(* Logix 5000 project; controller BTS01 vendor 1 type 14 code 217 rev 32.14; software revision 32.04; part 11 of 15 *)
(* tags used below, declared in another part *)
   AG1101 : DTE_VFD;   // Tank 1100 Agitator
   AG1101_CIP_ENABLE : BOOL;
   AG1201 : DTE_VFD;   // Tank 1200 Agitator
   AG1201_CIP_ENABLE : BOOL;
   C02S01 : REAL[8];   // 5069-IF8
   C02S03 : INT;   // 5069-IB16
   C02S06 : INT;   // 5069-IB16
   CAUSTIC1_TIME_REM : DINT;   // CIP 1 CAUSTIC TIM REMAINING
   CIP1_SUPPLY_TEMP_OFFSET : DINT;   // CIP 1 SUPPLY TEMP OFFSET FROM RETURN TEMP SETPOINT
   CIP_1_ACTIVE_CIRCUIT : DINT;
   CIP_1_ACTIVE_PROGRAM : CIP_PROGRAM;
   CIP_1_ACTIVE_STEP : CIP_STEP_DEF;   // CIP 1 ACTIVE STEP DATA
   CIP_1_ACTIVE_STEP_NUMBER : DINT;
   CIP_1_ACTIVE_STEP_SUP_TEMP : DINT;   // CIP 1 SUPPLY TEMP SETPOINT FOR ACTIVE STEP
   CIP_1_ACTIVE_STEP_TIME : DINT;
   CIP_1_ALARM_INDICATOR : DINT;   // ALARM STATE INDICATOR AT HMI
   CIP_1_ALARMS : DINT[30];
   CIP_1_CAUSTIC_TRANS_ACT : BOOL;   // CIP 1 RETURN TO CAUSTIC TANK LEVEL TRANSITION ACTIVE
   CIP_1_CIRCUIT_SELECT_HMI : INT;
   CIP_1_CURRENT_STEP_MESSAGE_INT : DINT;
   CIP_1_FLOW_PROOF : BOOL;   // CIP 1 FLOW PROOF BIT 0 = NO FLOW 1 = FLOW
   CIP_1_HOLD_LATCH : BOOL;
   CIP_1_HOLD_PB_CTU : COUNTER;
   CIP_1_HOLD_PB_HMI : BOOL;
   CIP_1_HOLD_TIME : REAL;
   CIP_1_LOAD_ACTIVE_CIP_RECIPE_PB : BOOL;
   CIP_1_OPERATOR_ACK : BOOL;   // CIP 1 SEQUENCER OPERATOR ACKNOWLEDGE
   CIP_1_OPERATOR_ACK_PB_HMI : BOOL;
   CIP_1_PRERINSE_TRANS_ACT : BOOL;   // CIP 1 RETURN TO PRERINSE TANK LEVEL TRANSITION ACTIVE
   CIP_1_PROGRAMS : CIP_PROGRAM[30];
   CIP_1_RECIPE_SELECTED_HMI : STRING;
   CIP_1_RESET_PB_HMI : BOOL;
   CIP_1_RUN_LATCH : BOOL;
   CIP_1_SANITIZE_SEL_PB : BOOL;   // CIP 1 SANITIZE ONLY HMI SELECT PB 0 = FULL CIP CYCLE 1 = SANITIZE ONLY
   CIP_1_SECONDS : DINT;   // CIP 1 SECONDS REMAINING IN MINUTE
   CIP_1_SECONDS_REMAINING : DINT;
   CIP_1_SEQ_CTU : COUNTER;   // CIP 1 SEQUENCE STEP COUNTER THIS IS THE SEQUENCE STEP CONTROL
   CIP_1_SEQ_ENABLE : DINT;   // CIP 1 SEQUENCER DATA TO BE ENABLED FOR OPERATION DURING CIP
   CIP_1_SEQ_MEMORY_REG : DINT;
   CIP_1_START_PB_HMI : BOOL;
   CIP_1_STEP_ADV_ACTIVE : BOOL;   // CIP 1 SEQUENCER STEP ADVANCE ACTIVE
   CIP_1_STEP_ADV_MESSAGE : BOOL;
   CIP_1_STEP_ADV_MESSAGE_INT : DINT;
   CIP_1_STEP_ADVANCE : BOOL;   // CIP 1 SEQUENCER MANUAL STEP ADVANCE
   CIP_1_STEP_ADVANCE_PB_HMI : BOOL;
   CIP_1_STOP_DURING_RUN : BOOL;   // CIP 1 SEQUENCER STOPPED DURING RUN
   CIP_1_STOP_PB_HMI : BOOL;
   CIP_1_SUPPLY_TEMP_SPT : DINT;   // CIP 1 SUPPLY TEMP SETPOINT
   CIP_1_TIME_ELAPSED_MIN : DINT;
   CIP_1_TIME_ELAPSED_SEC : DINT;
   CIP_1_TIME_REMAINING : REAL;
   CIP_1_TIME_REMAINING_MINR : DINT;   // TIME REMAINING IN MINUTES TO HMI
   CIP_1_TIME_REMAINING_SECR : DINT;   // TIME REMAINING IN SECONDS TO HMI
   CIP_RinseStep_PULSE_ENABLE : BOOL;
   CIP_SUPPLY_PUMP_CIP_ENABLE : BOOL;
   CIP_WashStep_PULSE_ENABLE : BOOL;
   DTE_TEST : DINT;   // TEST CIP BIT REMOVE WHEN FULL CIP CODE HAS BEEN COMPLETED ==================== Always True Bit
   HMI_Operator_Ack_REQUEST : BOOL;   // CIP 1 Operator Acknowledge Request Active to Proceed to Next Step
   Message_Visibility_1 : DINT;
   OK_TO_PROCEED_PB_HMI : BOOL;
   OK_TO_PROCEED_PB_TIMER : TIMER;
   ONS : DINT[20];   // ONE_SHOT_BIT
   P1001_CIP_Enable : BOOL;
   P1002_CIP_ENABLE : BOOL;
   P1003_CIP_ENABLE : BOOL;
   PRE_RINSE_TANK_LEVEL_OFF_PERC : DINT;   // HMI INPUT OF WATER LEVEL OFF IN %
   PRERINSE_TIME_REM : DINT;   // PRERINSE TIME REMAINING
   SANITIZE_ENABLE_TRIGGER : BOOL;   // ADVANCE TRIGGER TO NEXT SANITIZE STEP
   STEP_TIME_MIN : DINT;   // CIP 1 STEP TIMER CONTROLS TIMING PRESET FOR EACH TIMED STEP TO HMI
   STEP_TIME_SEC : DINT;   // CIP 1 STEP TIMER CONTROLS TIMING PRESET FOR EACH TIMED STEP TO HMI
   TIMERS : TIMER[30];
   TOTALIZER_MIN : DINT;   // CIP 1 TOTALIZER (MIN)
   TOTALIZER_SEC : DINT;   // CIP 1 TOTALIZER (SEC)
   TransferEnabled : BOOL;
   TransferSelected : DINT;
   UnloadEnabled : BOOL;
   UnloadSelected : DINT;
   V1001_CIP_ENABLE : BOOL;
   V1002 : DTE_Air_Valve_v2;   // CIP Bypass Valve
   V1002_CIP_ENABLE : BOOL;
   V1003 : DTE_Air_Valve_v2;   // Filler Valve
   V1003_CIP_ENABLE : BOOL;
   V1004 : DTE_Air_Valve_v2;   // Filler Valve
   V1004_CIP_ENABLE : BOOL;
   V1005 : DTE_Air_Valve_v2;   // Filler Valve
   V1005_CIP_ENABLE : BOOL;
   V1006 : DTE_Air_Valve_v2;   // Filler Valve
   V1006_CIP_ENABLE : BOOL;
   V1007 : DTE_Air_Valve_v2;   // Filler Valve
   V1007_CIP_ENABLE : BOOL;
   V1101 : DTE_Air_Valve_v2;   // Tank 1100 Fill Valve
   V1101_CIP_ENABLE : BOOL;
   V1102 : DTE_Air_Valve_v2;   // Tank 1100 Discharge Valve
   V1102_CIP_ENABLE : BOOL;
   V1103 : DTE_Air_Valve_v2;   // Tank 1100 Line Valve
   V1103_CIP_ENABLE : BOOL;
   V1201 : DTE_Air_Valve_v2;   // Tank 1200 Fill Valve
   V1201_CIP_ENABLE : BOOL;
   V1202 : DTE_Air_Valve_v2;   // Tank 1200 Discharge Valve
   V1202_CIP_ENABLE : BOOL;
   V1203 : DTE_Air_Valve_v2;   // Tank 1200 Line Valve
   V1203_CIP_ENABLE : BOOL;

PROGRAM CIP   (* main routine Main_Routine *)

ROUTINE CIP_Control   (* ladder *)
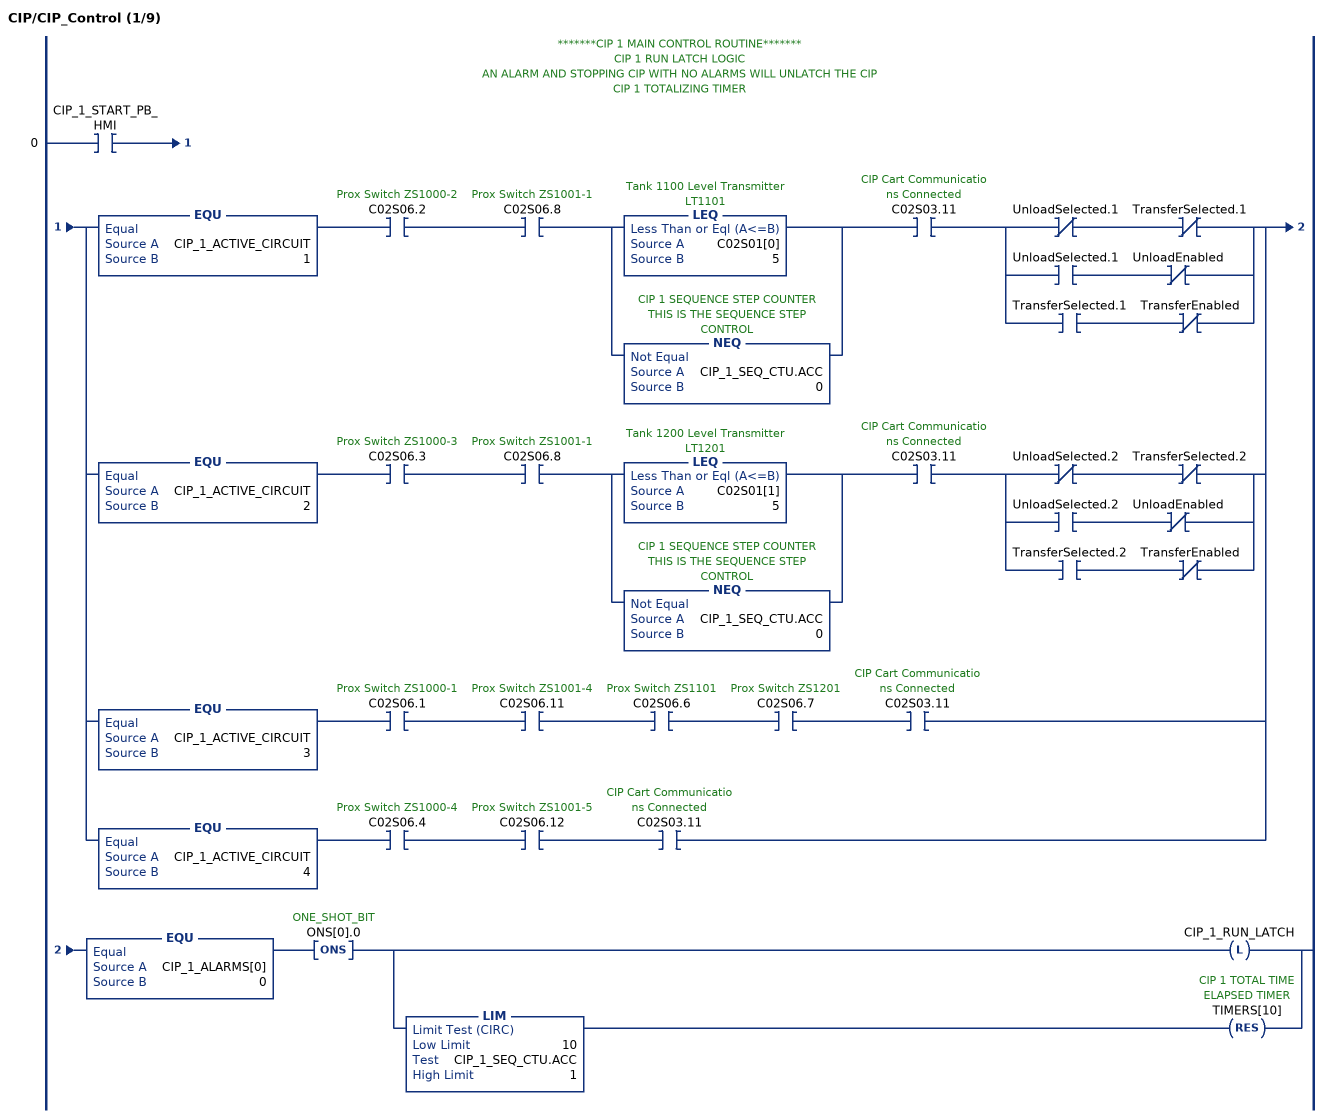
   // *******CIP 1 MAIN CONTROL ROUTINE*******
   // CIP 1 RUN LATCH LOGIC
   // AN ALARM AND STOPPING CIP WITH NO ALARMS WILL UNLATCH THE CIP
   // CIP 1 TOTALIZING TIMER
   0: XIC(CIP_1_START_PB_HMI)[EQU(CIP_1_ACTIVE_CIRCUIT,1) XIC(C02S06.2) XIC(C02S06.8) [LEQ(C02S01[0],5) ,NEQ(CIP_1_SEQ_CTU.ACC,0) ] XIC(C02S03.11) [XIO(UnloadSelected.1) XIO(TransferSelected.1) ,XIC(UnloadSelected.1) XIO(UnloadEnabled) ,XIC(TransferSelected.1) XIO(TransferEnabled) ] ,EQU(CIP_1_ACTIVE_CIRCUIT,2) XIC(C02S06.3) XIC(C02S06.8) [LEQ(C02S01[1],5) ,NEQ(CIP_1_SEQ_CTU.ACC,0) ] XIC(C02S03.11) [XIO(UnloadSelected.2) XIO(TransferSelected.2) ,XIC(UnloadSelected.2) XIO(UnloadEnabled) ,XIC(TransferSelected.2) XIO(TransferEnabled) ] ,EQU(CIP_1_ACTIVE_CIRCUIT,3) XIC(C02S06.1) XIC(C02S06.11) XIC(C02S06.6) XIC(C02S06.7) XIC(C02S03.11) ,EQU(CIP_1_ACTIVE_CIRCUIT,4) XIC(C02S06.4) XIC(C02S06.12) XIC(C02S03.11) ]EQU(CIP_1_ALARMS[0],0)ONS(ONS[0].0)[OTL(CIP_1_RUN_LATCH) ,LIM(10,CIP_1_SEQ_CTU.ACC,1) RES(TIMERS[10]) ];
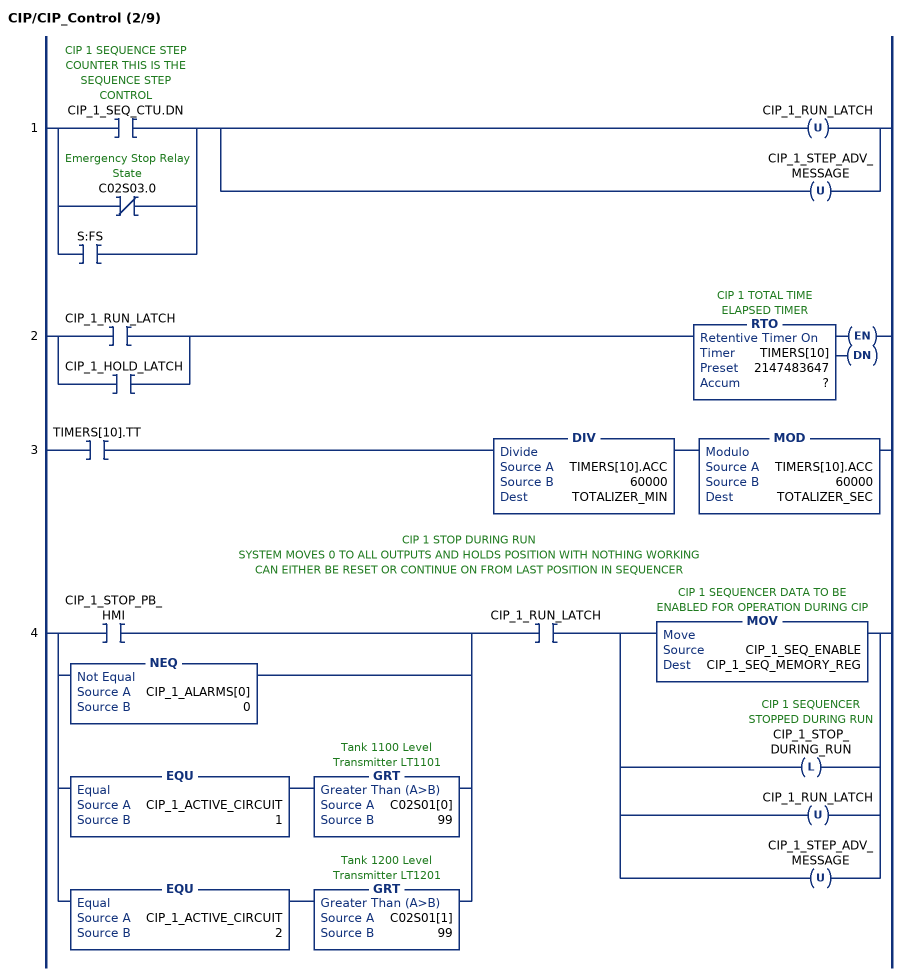
   1: [XIC(CIP_1_SEQ_CTU.DN) ,XIO(C02S03.0) ,XIC(S:FS) ][OTU(CIP_1_RUN_LATCH) ,OTU(CIP_1_STEP_ADV_MESSAGE) ];
   2: [XIC(CIP_1_RUN_LATCH) ,XIC(CIP_1_HOLD_LATCH) ]RTO(TIMERS[10],?,?);
   3: XIC(TIMERS[10].TT)DIV(TIMERS[10].ACC,60000,TOTALIZER_MIN)MOD(TIMERS[10].ACC,60000,TOTALIZER_SEC);
   // CIP 1 STOP DURING RUN
   // SYSTEM MOVES 0 TO ALL OUTPUTS AND HOLDS POSITION WITH NOTHING WORKING
   // CAN EITHER BE RESET OR CONTINUE ON FROM LAST POSITION IN SEQUENCER
   4: [XIC(CIP_1_STOP_PB_HMI) ,NEQ(CIP_1_ALARMS[0],0) ,EQU(CIP_1_ACTIVE_CIRCUIT,1) GRT(C02S01[0],99) ,EQU(CIP_1_ACTIVE_CIRCUIT,2) GRT(C02S01[1],99) ]XIC(CIP_1_RUN_LATCH)[MOV(CIP_1_SEQ_ENABLE,CIP_1_SEQ_MEMORY_REG) ,OTL(CIP_1_STOP_DURING_RUN) ,OTU(CIP_1_RUN_LATCH) ,OTU(CIP_1_STEP_ADV_MESSAGE) ];
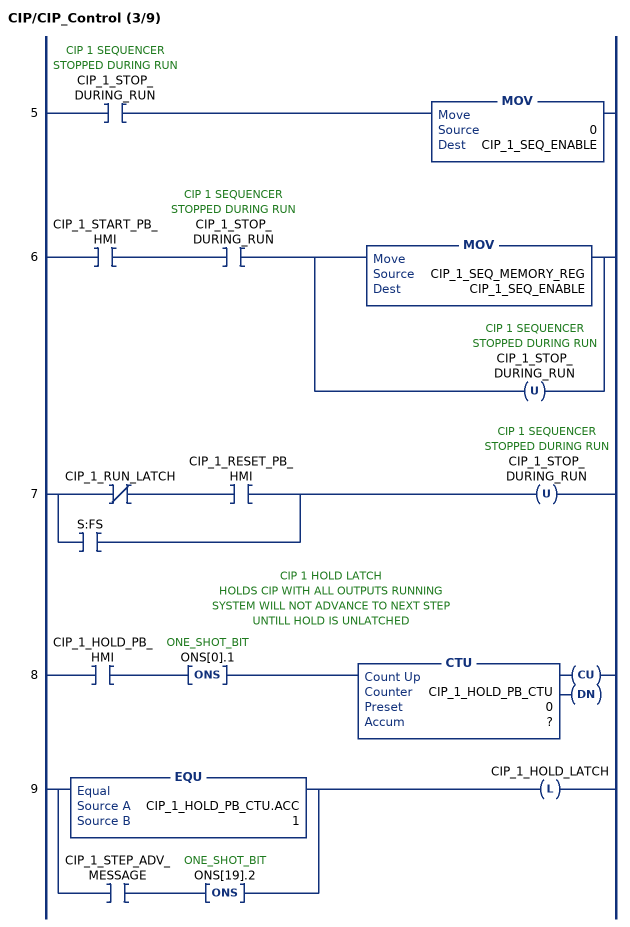
   5: XIC(CIP_1_STOP_DURING_RUN)MOV(0,CIP_1_SEQ_ENABLE);
   6: XIC(CIP_1_START_PB_HMI)XIC(CIP_1_STOP_DURING_RUN)[MOV(CIP_1_SEQ_MEMORY_REG,CIP_1_SEQ_ENABLE) ,OTU(CIP_1_STOP_DURING_RUN) ];
   7: [XIO(CIP_1_RUN_LATCH) XIC(CIP_1_RESET_PB_HMI) ,XIC(S:FS) ]OTU(CIP_1_STOP_DURING_RUN);
   // CIP 1 HOLD LATCH
   // HOLDS CIP WITH ALL OUTPUTS RUNNING
   // SYSTEM WILL NOT ADVANCE TO NEXT STEP
   // UNTILL HOLD IS UNLATCHED
   8: XIC(CIP_1_HOLD_PB_HMI)ONS(ONS[0].1)CTU(CIP_1_HOLD_PB_CTU,?,?);
   9: [EQU(CIP_1_HOLD_PB_CTU.ACC,1) ,XIC(CIP_1_STEP_ADV_MESSAGE) ONS(ONS[19].2) ]OTL(CIP_1_HOLD_LATCH);
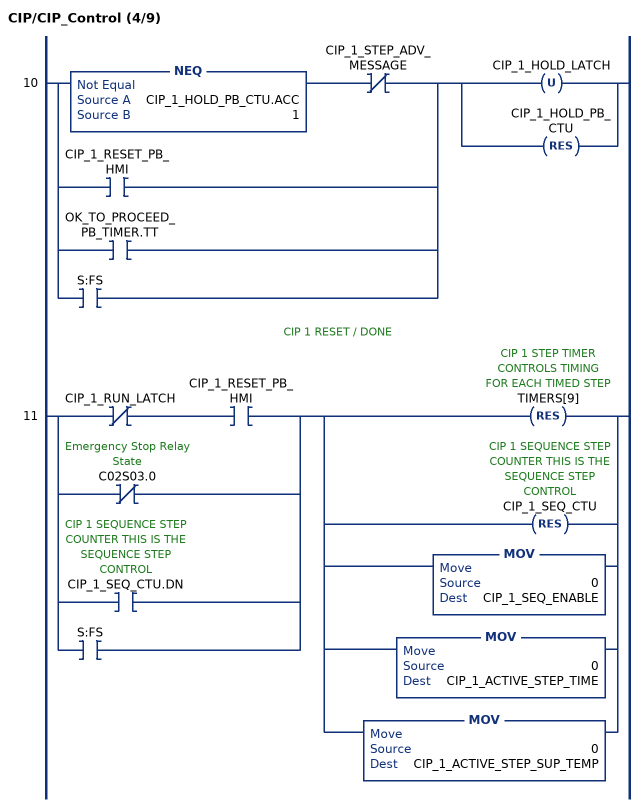
   10: [NEQ(CIP_1_HOLD_PB_CTU.ACC,1) XIO(CIP_1_STEP_ADV_MESSAGE) ,XIC(CIP_1_RESET_PB_HMI) ,XIC(OK_TO_PROCEED_PB_TIMER.TT) ,XIC(S:FS) ][OTU(CIP_1_HOLD_LATCH) ,RES(CIP_1_HOLD_PB_CTU) ];
   // CIP 1 RESET / DONE
   11: [XIO(CIP_1_RUN_LATCH) XIC(CIP_1_RESET_PB_HMI) ,XIO(C02S03.0) ,XIC(CIP_1_SEQ_CTU.DN) ,XIC(S:FS) ][RES(TIMERS[9]) ,RES(CIP_1_SEQ_CTU) ,MOV(0,CIP_1_SEQ_ENABLE) ,MOV(0,CIP_1_ACTIVE_STEP_TIME) ,MOV(0,CIP_1_ACTIVE_STEP_SUP_TEMP) ];
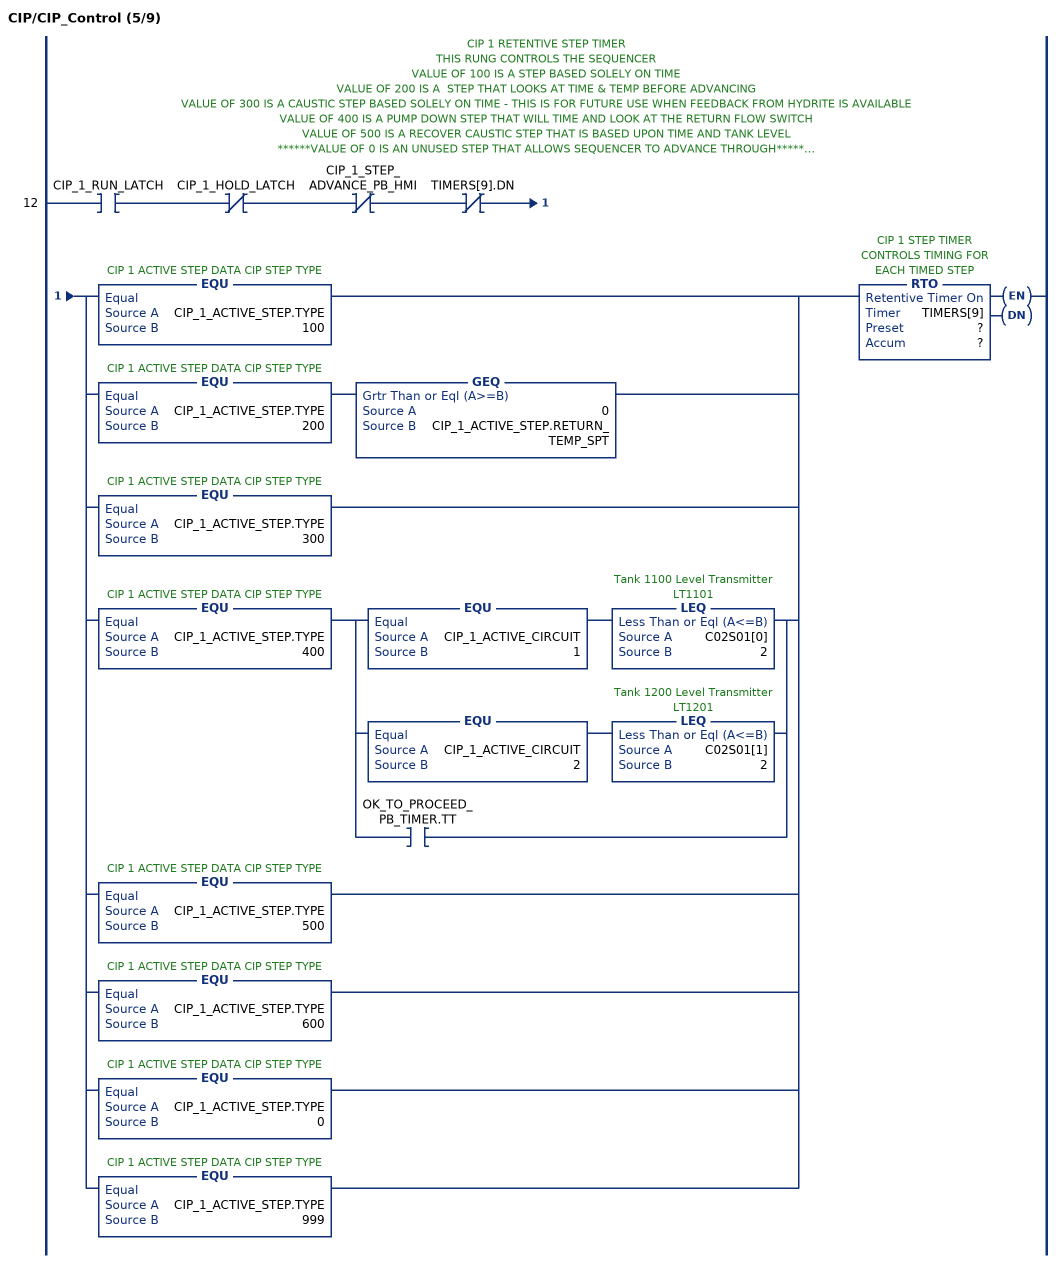
   // CIP 1 RETENTIVE STEP TIMER
   // THIS RUNG CONTROLS THE SEQUENCER
   // VALUE OF 100 IS A STEP BASED SOLELY ON TIME
   // VALUE OF 200 IS A  STEP THAT LOOKS AT TIME & TEMP BEFORE ADVANCING
   // VALUE OF 300 IS A CAUSTIC STEP BASED SOLELY ON TIME - THIS IS FOR FUTURE USE WHEN FEEDBACK FROM HYDRITE IS AVAILABLE
   // VALUE OF 400 IS A PUMP DOWN STEP THAT WILL TIME AND LOOK AT THE RETURN FLOW SWITCH
   // VALUE OF 500 IS A RECOVER CAUSTIC STEP THAT IS BASED UPON TIME AND TANK LEVEL
   // ******VALUE OF 0 IS AN UNUSED STEP THAT ALLOWS SEQUENCER TO ADVANCE THROUGH******
   // 999 IS THE LAST STEP OF THE PROGRAM AND IS AN UNUSED STEP
   12: XIC(CIP_1_RUN_LATCH)XIO(CIP_1_HOLD_LATCH)XIO(CIP_1_STEP_ADVANCE_PB_HMI)XIO(TIMERS[9].DN)[EQU(CIP_1_ACTIVE_STEP.TYPE,100) ,EQU(CIP_1_ACTIVE_STEP.TYPE,200) GEQ(0,CIP_1_ACTIVE_STEP.RETURN_TEMP_SPT) ,EQU(CIP_1_ACTIVE_STEP.TYPE,300) ,EQU(CIP_1_ACTIVE_STEP.TYPE,400) [EQU(CIP_1_ACTIVE_CIRCUIT,1) LEQ(C02S01[0],2) ,EQU(CIP_1_ACTIVE_CIRCUIT,2) LEQ(C02S01[1],2) ,XIC(OK_TO_PROCEED_PB_TIMER.TT) ] ,EQU(CIP_1_ACTIVE_STEP.TYPE,500) ,EQU(CIP_1_ACTIVE_STEP.TYPE,600) ,[EQU(CIP_1_ACTIVE_STEP.TYPE,0) ,EQU(CIP_1_ACTIVE_STEP.TYPE,999) ] ]RTO(TIMERS[9],?,?);
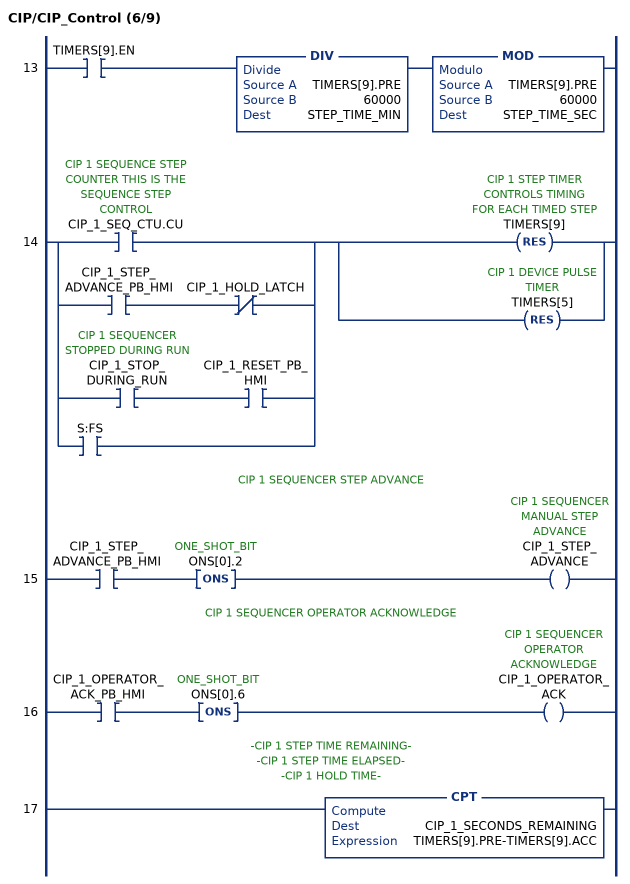
   13: XIC(TIMERS[9].EN)DIV(TIMERS[9].PRE,60000,STEP_TIME_MIN)MOD(TIMERS[9].PRE,60000,STEP_TIME_SEC);
   14: [XIC(CIP_1_SEQ_CTU.CU) ,XIC(CIP_1_STEP_ADVANCE_PB_HMI) XIO(CIP_1_HOLD_LATCH) ,XIC(CIP_1_STOP_DURING_RUN) XIC(CIP_1_RESET_PB_HMI) ,XIC(S:FS) ][RES(TIMERS[9]) ,RES(TIMERS[5]) ];
   // CIP 1 SEQUENCER STEP ADVANCE
   15: XIC(CIP_1_STEP_ADVANCE_PB_HMI)ONS(ONS[0].2)OTE(CIP_1_STEP_ADVANCE);
   // CIP 1 SEQUENCER OPERATOR ACKNOWLEDGE
   16: XIC(CIP_1_OPERATOR_ACK_PB_HMI)ONS(ONS[0].6)OTE(CIP_1_OPERATOR_ACK);
   // -CIP 1 STEP TIME REMAINING-
   // -CIP 1 STEP TIME ELAPSED-
   // -CIP 1 HOLD TIME-
   17: CPT(CIP_1_SECONDS_REMAINING,TIMERS[9].PRE-TIMERS[9].ACC);
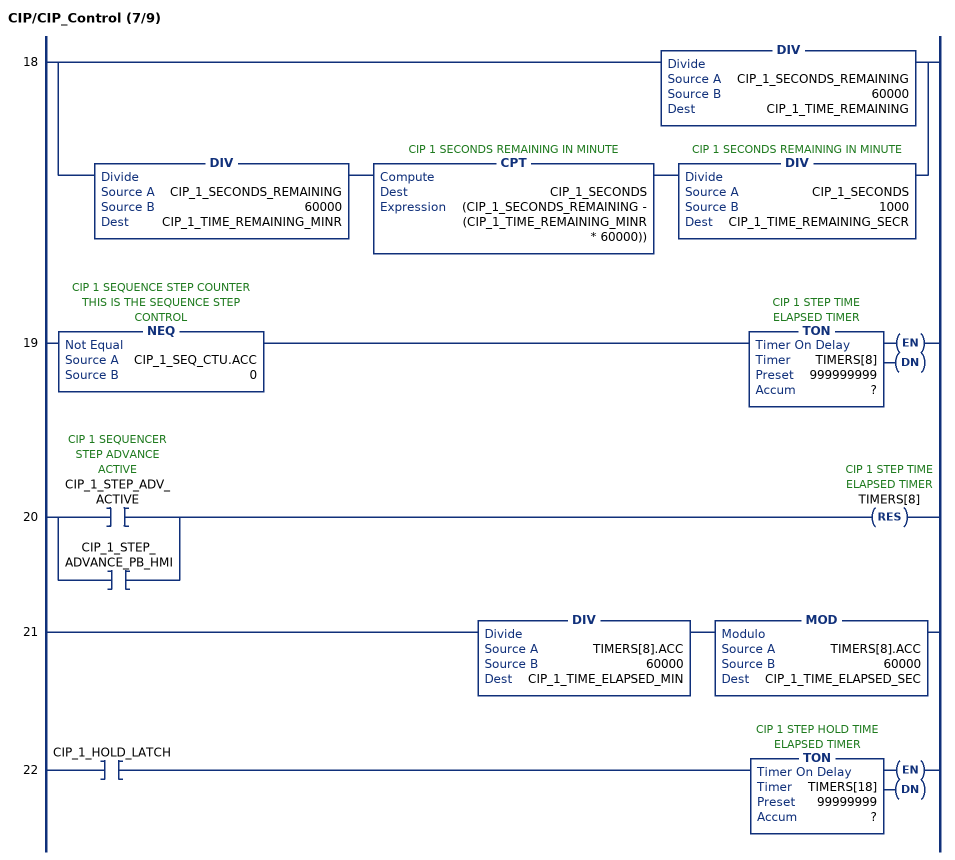
   18: [DIV(CIP_1_SECONDS_REMAINING,60000,CIP_1_TIME_REMAINING) ,DIV(CIP_1_SECONDS_REMAINING,60000,CIP_1_TIME_REMAINING_MINR) CPT(CIP_1_SECONDS,(CIP_1_SECONDS_REMAINING - (CIP_1_TIME_REMAINING_MINR * 60000))) DIV(CIP_1_SECONDS,1000,CIP_1_TIME_REMAINING_SECR) ];
   19: NEQ(CIP_1_SEQ_CTU.ACC,0)TON(TIMERS[8],?,?);
   20: [XIC(CIP_1_STEP_ADV_ACTIVE) ,XIC(CIP_1_STEP_ADVANCE_PB_HMI) ]RES(TIMERS[8]);
   21: DIV(TIMERS[8].ACC,60000,CIP_1_TIME_ELAPSED_MIN)MOD(TIMERS[8].ACC,60000,CIP_1_TIME_ELAPSED_SEC);
   22: XIC(CIP_1_HOLD_LATCH)TON(TIMERS[18],?,?);
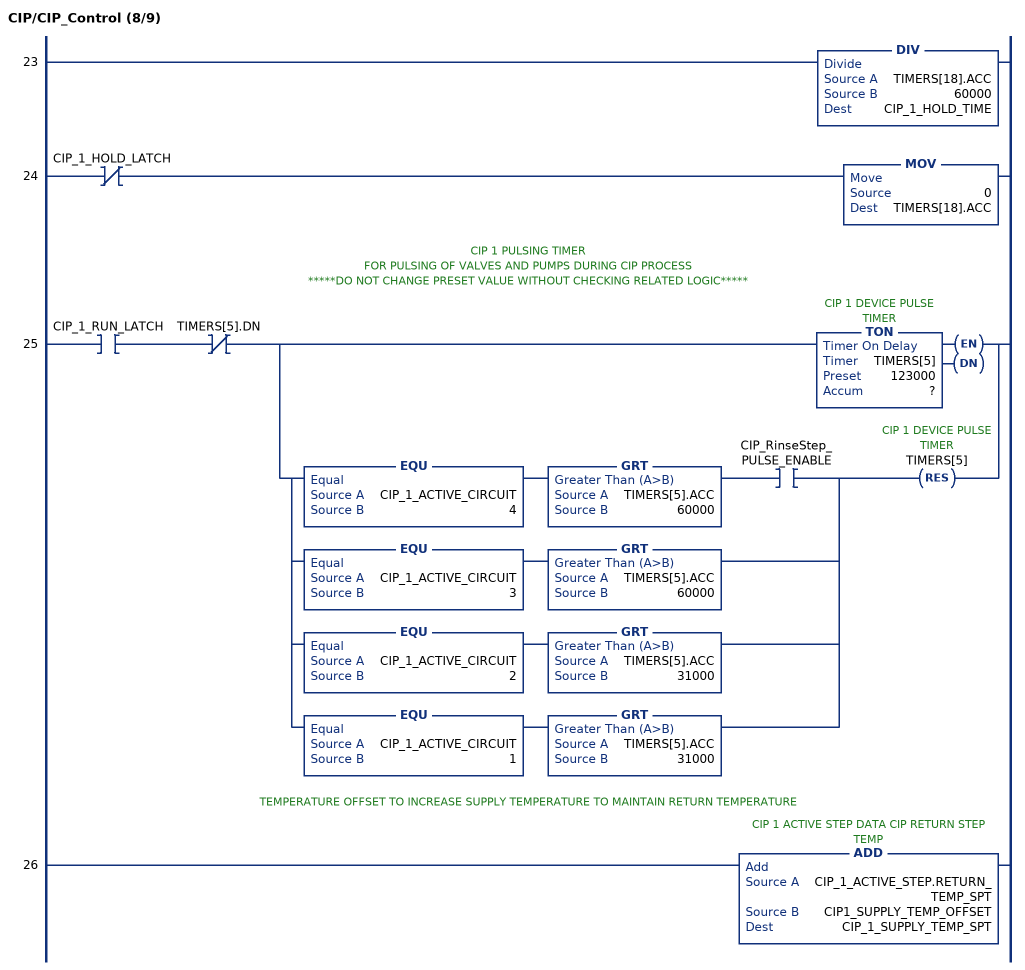
   23: DIV(TIMERS[18].ACC,60000,CIP_1_HOLD_TIME);
   24: XIO(CIP_1_HOLD_LATCH)MOV(0,TIMERS[18].ACC);
   // CIP 1 PULSING TIMER
   // FOR PULSING OF VALVES AND PUMPS DURING CIP PROCESS
   // *****DO NOT CHANGE PRESET VALUE WITHOUT CHECKING RELATED LOGIC*****
   25: XIC(CIP_1_RUN_LATCH)XIO(TIMERS[5].DN)[TON(TIMERS[5],?,?) ,[EQU(CIP_1_ACTIVE_CIRCUIT,4) GRT(TIMERS[5].ACC,60000) XIC(CIP_RinseStep_PULSE_ENABLE) ,EQU(CIP_1_ACTIVE_CIRCUIT,3) GRT(TIMERS[5].ACC,60000) ,EQU(CIP_1_ACTIVE_CIRCUIT,2) GRT(TIMERS[5].ACC,31000) ,EQU(CIP_1_ACTIVE_CIRCUIT,1) GRT(TIMERS[5].ACC,31000) ] RES(TIMERS[5]) ];
   // TEMPERATURE OFFSET TO INCREASE SUPPLY TEMPERATURE TO MAINTAIN RETURN TEMPERATURE
   26: ADD(CIP_1_ACTIVE_STEP.RETURN_TEMP_SPT,CIP1_SUPPLY_TEMP_OFFSET,CIP_1_SUPPLY_TEMP_SPT);
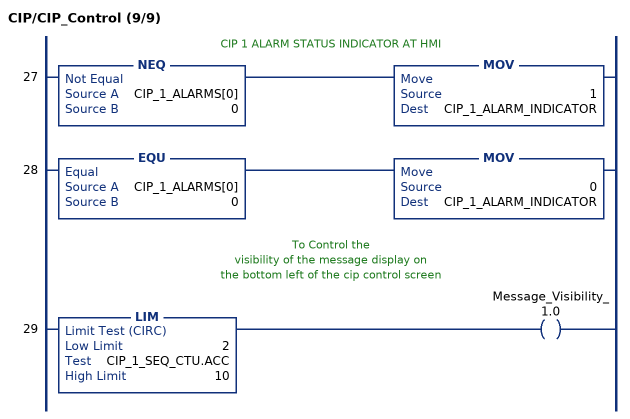
   // CIP 1 ALARM STATUS INDICATOR AT HMI
   27: NEQ(CIP_1_ALARMS[0],0)MOV(1,CIP_1_ALARM_INDICATOR);
   28: EQU(CIP_1_ALARMS[0],0)MOV(0,CIP_1_ALARM_INDICATOR);
   // To Control the
   // visibility of the message display on
   // the bottom left of the cip control screen
   29: LIM(2,CIP_1_SEQ_CTU.ACC,10)OTE(Message_Visibility_1.0);
END_ROUTINE

ROUTINE CIP_Program_Select   (* ladder *)
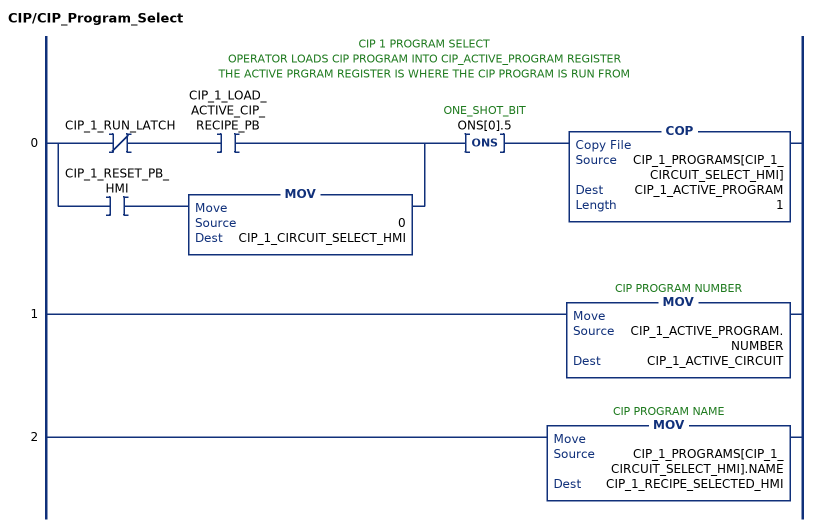
   // CIP 1 PROGRAM SELECT
   // OPERATOR LOADS CIP PROGRAM INTO CIP_ACTIVE_PROGRAM REGISTER
   // THE ACTIVE PRGRAM REGISTER IS WHERE THE CIP PROGRAM IS RUN FROM
   0: [XIO(CIP_1_RUN_LATCH) XIC(CIP_1_LOAD_ACTIVE_CIP_RECIPE_PB) ,XIC(CIP_1_RESET_PB_HMI) MOV(0,CIP_1_CIRCUIT_SELECT_HMI) ]ONS(ONS[0].5)COP(CIP_1_PROGRAMS[CIP_1_CIRCUIT_SELECT_HMI],CIP_1_ACTIVE_PROGRAM,1);
   1: MOV(CIP_1_ACTIVE_PROGRAM.NUMBER,CIP_1_ACTIVE_CIRCUIT);
   2: MOV(CIP_1_PROGRAMS[CIP_1_CIRCUIT_SELECT_HMI].NAME,CIP_1_RECIPE_SELECTED_HMI);
END_ROUTINE

ROUTINE CIP_Sequencer   (* ladder *)
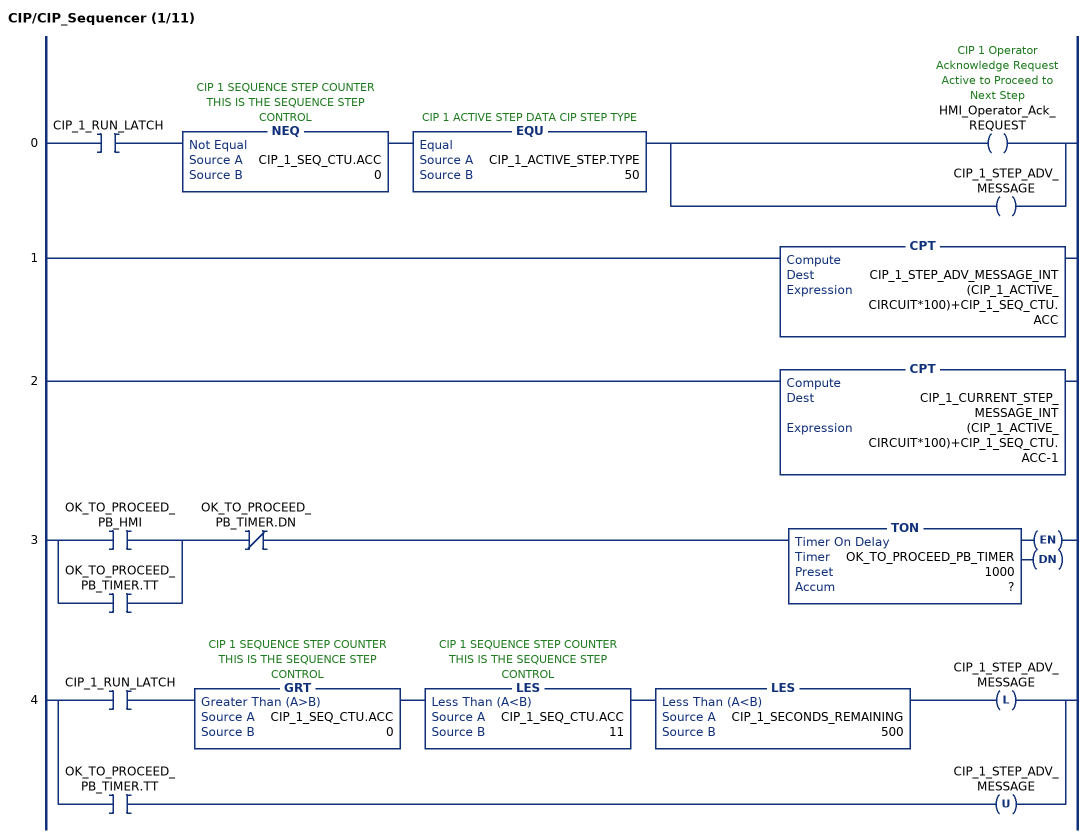
   0: XIC(CIP_1_RUN_LATCH)NEQ(CIP_1_SEQ_CTU.ACC,0)EQU(CIP_1_ACTIVE_STEP.TYPE,50)[OTE(HMI_Operator_Ack_REQUEST) ,OTE(CIP_1_STEP_ADV_MESSAGE) ];
   1: CPT(CIP_1_STEP_ADV_MESSAGE_INT,(CIP_1_ACTIVE_CIRCUIT*100)+CIP_1_SEQ_CTU.ACC);
   2: CPT(CIP_1_CURRENT_STEP_MESSAGE_INT,(CIP_1_ACTIVE_CIRCUIT*100)+CIP_1_SEQ_CTU.ACC-1);
   3: [XIC(OK_TO_PROCEED_PB_HMI) ,XIC(OK_TO_PROCEED_PB_TIMER.TT) ]XIO(OK_TO_PROCEED_PB_TIMER.DN)TON(OK_TO_PROCEED_PB_TIMER,?,?);
   4: [XIC(CIP_1_RUN_LATCH) GRT(CIP_1_SEQ_CTU.ACC,0) LES(CIP_1_SEQ_CTU.ACC,11) LES(CIP_1_SECONDS_REMAINING,500) OTL(CIP_1_STEP_ADV_MESSAGE) ,XIC(OK_TO_PROCEED_PB_TIMER.TT) OTU(CIP_1_STEP_ADV_MESSAGE) ];
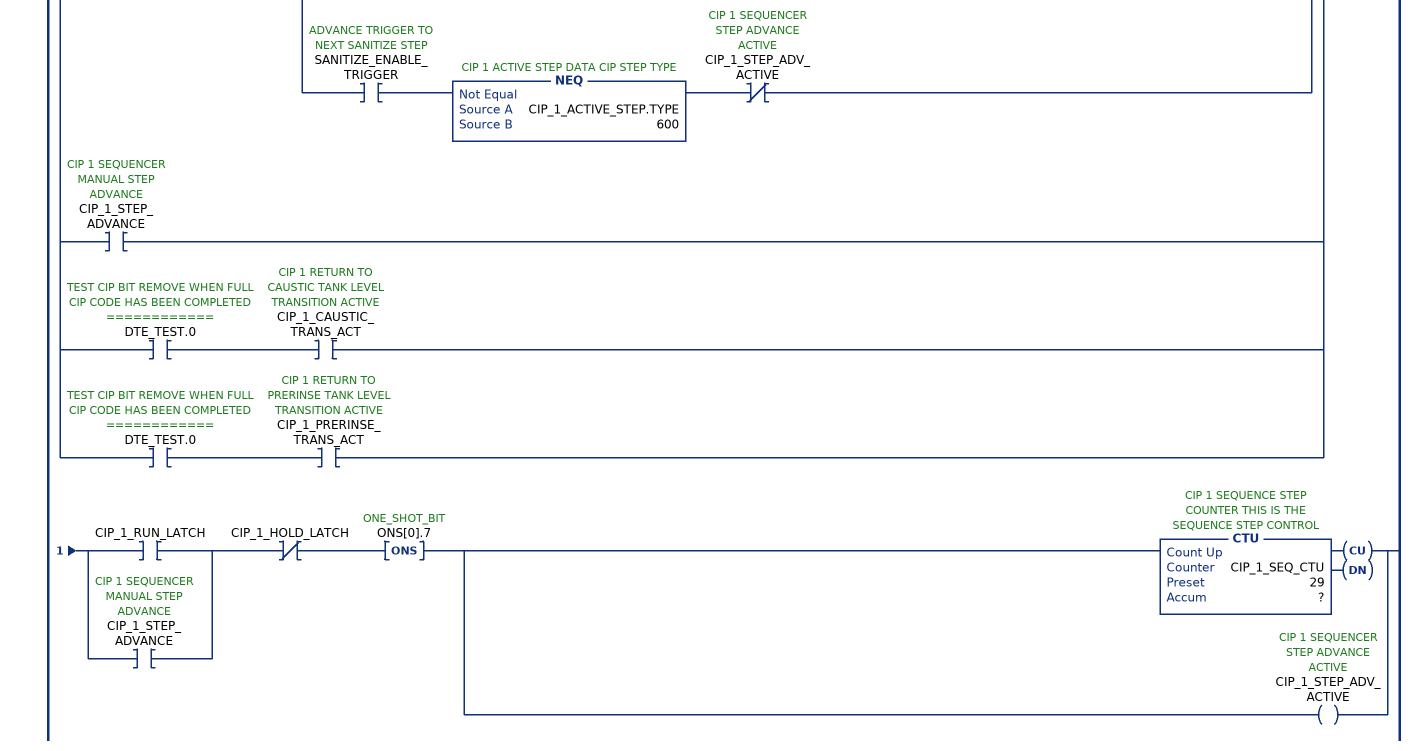
   // CIP 1 SEQUENCER ADVANCE LOGIC
   // THE STEPS WILL ADVANCE WHEN:
   // 1.  THE STEP TIMER IS DONE OR
   // 2.  THE STEP ADVANCE PB ON THE HMI HAS BEEN PRESSED OR
   // 3.  IF THE STEP TRANSITION BASED UPON TANK LEVEL IS ACTIVE
   // 4.  IF THE ACID STEP ENABLE BIT IS TRUE AND THE ACID PROGRAM ENABLE PB FROM HMI IS TRUE
   5: [EQU(CIP_1_SEQ_CTU.ACC,0) ,NEQ(CIP_1_SEQ_CTU.ACC,0) [EQU(CIP_1_ACTIVE_STEP.TYPE,50) [XIC(CIP_1_OPERATOR_ACK) ,XIC(OK_TO_PROCEED_PB_TIMER.TT) ] ,EQU(CIP_1_ACTIVE_STEP.TYPE,400) [XIC(TIMERS[9].DN) ,XIC(DTE_TEST.0) XIO(CIP_1_FLOW_PROOF) ] ,EQU(CIP_1_ACTIVE_STEP.TYPE,500) [XIC(TIMERS[9].DN) ,XIC(DTE_TEST.0) GEQ(100,PRE_RINSE_TANK_LEVEL_OFF_PERC) ] ,EQU(CIP_1_ACTIVE_STEP.TYPE,600) XIC(TIMERS[9].DN) ,XIO(SANITIZE_ENABLE_TRIGGER) NEQ(CIP_1_ACTIVE_STEP.TYPE,50) NEQ(CIP_1_ACTIVE_STEP.TYPE,400) NEQ(CIP_1_ACTIVE_STEP.TYPE,500) XIC(TIMERS[9].DN) ,XIC(SANITIZE_ENABLE_TRIGGER) NEQ(CIP_1_ACTIVE_STEP.TYPE,600) XIO(CIP_1_STEP_ADV_ACTIVE) ] ,XIC(CIP_1_STEP_ADVANCE) ,XIC(DTE_TEST.0) XIC(CIP_1_CAUSTIC_TRANS_ACT) ,XIC(DTE_TEST.0) XIC(CIP_1_PRERINSE_TRANS_ACT) ][XIC(CIP_1_RUN_LATCH) ,XIC(CIP_1_STEP_ADVANCE) ]XIO(CIP_1_HOLD_LATCH)ONS(ONS[0].7)[CTU(CIP_1_SEQ_CTU,?,?) ,OTE(CIP_1_STEP_ADV_ACTIVE) ];
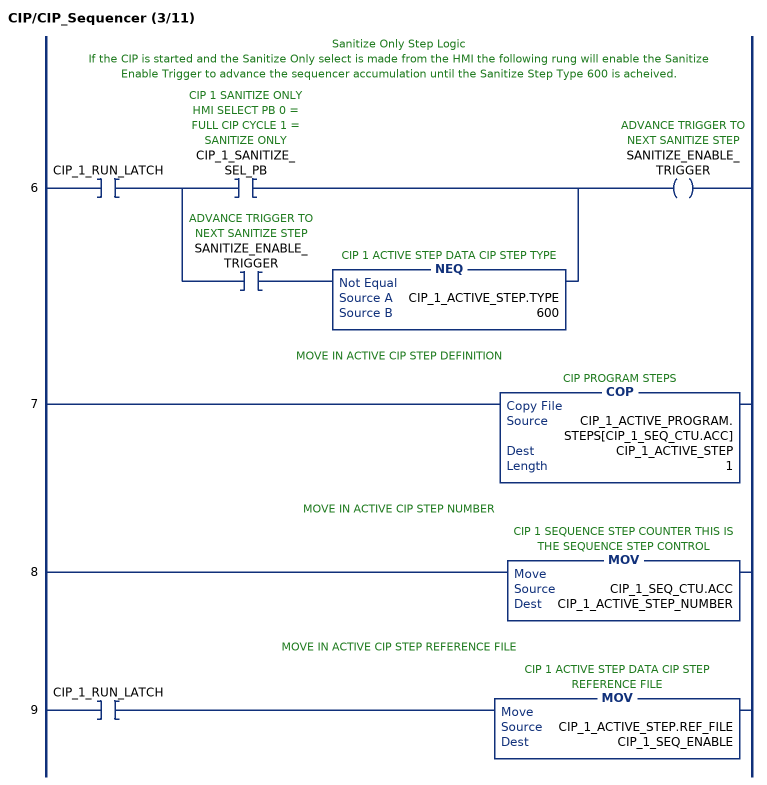
   // Sanitize Only Step Logic
   // If the CIP is started and the Sanitize Only select is made from the HMI the following rung will enable the Sanitize Enable Trigger to advance the sequencer accumulation until the Sanitize Step Type 600 is acheived.
   6: XIC(CIP_1_RUN_LATCH)[XIC(CIP_1_SANITIZE_SEL_PB) ,XIC(SANITIZE_ENABLE_TRIGGER) NEQ(CIP_1_ACTIVE_STEP.TYPE,600) ]OTE(SANITIZE_ENABLE_TRIGGER);
   // MOVE IN ACTIVE CIP STEP DEFINITION
   7: COP(CIP_1_ACTIVE_PROGRAM.STEPS[CIP_1_SEQ_CTU.ACC],CIP_1_ACTIVE_STEP,1);
   // MOVE IN ACTIVE CIP STEP NUMBER
   8: MOV(CIP_1_SEQ_CTU.ACC,CIP_1_ACTIVE_STEP_NUMBER);
   // MOVE IN ACTIVE CIP STEP REFERENCE FILE
   9: XIC(CIP_1_RUN_LATCH)MOV(CIP_1_ACTIVE_STEP.REF_FILE,CIP_1_SEQ_ENABLE);
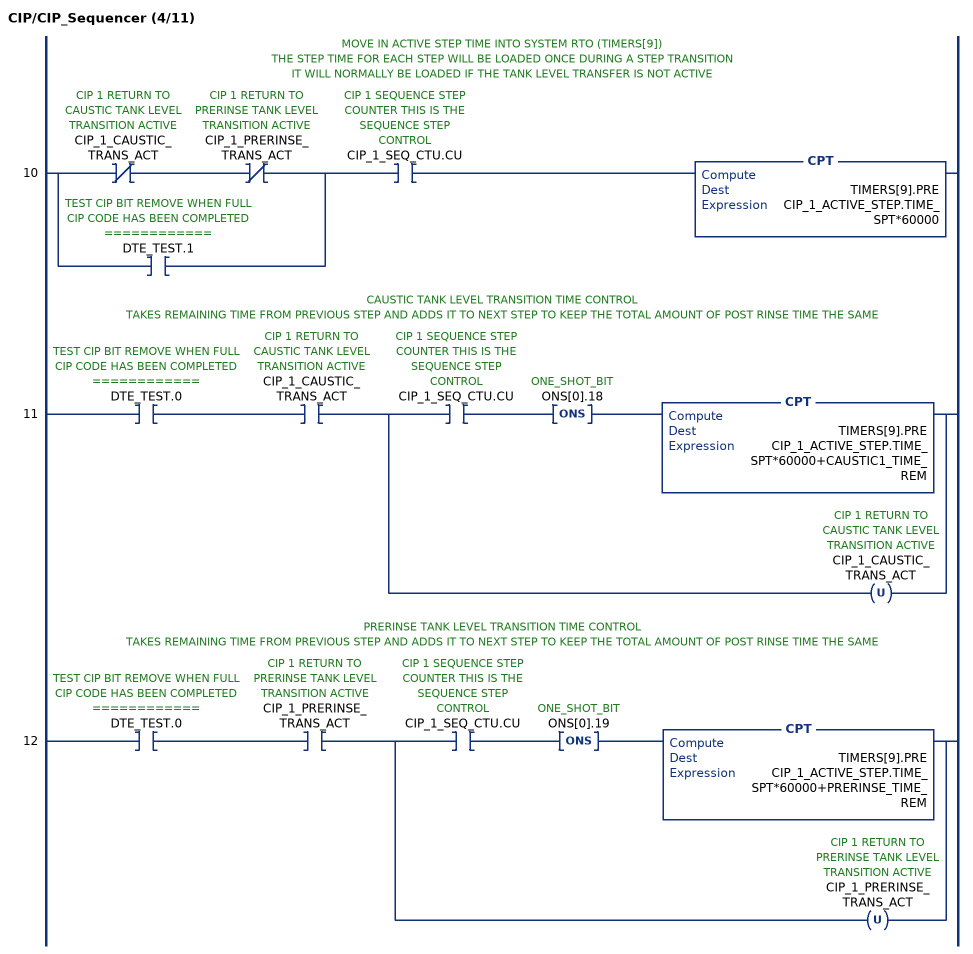
   // MOVE IN ACTIVE STEP TIME INTO SYSTEM RTO (TIMERS[9])
   // THE STEP TIME FOR EACH STEP WILL BE LOADED ONCE DURING A STEP TRANSITION
   // IT WILL NORMALLY BE LOADED IF THE TANK LEVEL TRANSFER IS NOT ACTIVE
   10: [XIO(CIP_1_CAUSTIC_TRANS_ACT) XIO(CIP_1_PRERINSE_TRANS_ACT) ,XIC(DTE_TEST.1) ]XIC(CIP_1_SEQ_CTU.CU)CPT(TIMERS[9].PRE,CIP_1_ACTIVE_STEP.TIME_SPT*60000);
   // CAUSTIC TANK LEVEL TRANSITION TIME CONTROL
   // TAKES REMAINING TIME FROM PREVIOUS STEP AND ADDS IT TO NEXT STEP TO KEEP THE TOTAL AMOUNT OF POST RINSE TIME THE SAME
   11: XIC(DTE_TEST.0)XIC(CIP_1_CAUSTIC_TRANS_ACT)[XIC(CIP_1_SEQ_CTU.CU) ONS(ONS[0].18) CPT(TIMERS[9].PRE,CIP_1_ACTIVE_STEP.TIME_SPT*60000+CAUSTIC1_TIME_REM) ,OTU(CIP_1_CAUSTIC_TRANS_ACT) ];
   // PRERINSE TANK LEVEL TRANSITION TIME CONTROL
   // TAKES REMAINING TIME FROM PREVIOUS STEP AND ADDS IT TO NEXT STEP TO KEEP THE TOTAL AMOUNT OF POST RINSE TIME THE SAME
   12: XIC(DTE_TEST.0)XIC(CIP_1_PRERINSE_TRANS_ACT)[XIC(CIP_1_SEQ_CTU.CU) ONS(ONS[0].19) CPT(TIMERS[9].PRE,CIP_1_ACTIVE_STEP.TIME_SPT*60000+PRERINSE_TIME_REM) ,OTU(CIP_1_PRERINSE_TRANS_ACT) ];
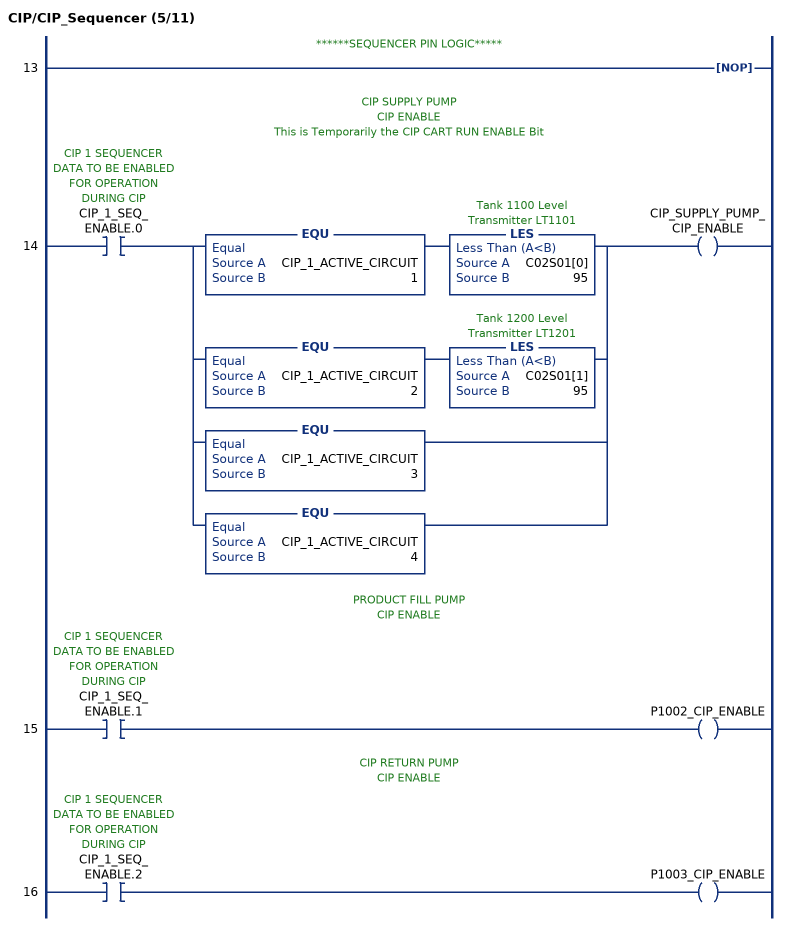
   // ******SEQUENCER PIN LOGIC*****
   13: NOP();
   // CIP SUPPLY PUMP
   // CIP ENABLE
   // This is Temporarily the CIP CART RUN ENABLE Bit
   14: XIC(CIP_1_SEQ_ENABLE.0)[EQU(CIP_1_ACTIVE_CIRCUIT,1) LES(C02S01[0],95) ,EQU(CIP_1_ACTIVE_CIRCUIT,2) LES(C02S01[1],95) ,EQU(CIP_1_ACTIVE_CIRCUIT,3) ,EQU(CIP_1_ACTIVE_CIRCUIT,4) ]OTE(CIP_SUPPLY_PUMP_CIP_ENABLE);
   // PRODUCT FILL PUMP
   // CIP ENABLE
   15: XIC(CIP_1_SEQ_ENABLE.1)OTE(P1002_CIP_ENABLE);
   // CIP RETURN PUMP
   // CIP ENABLE
   16: XIC(CIP_1_SEQ_ENABLE.2)OTE(P1003_CIP_ENABLE);
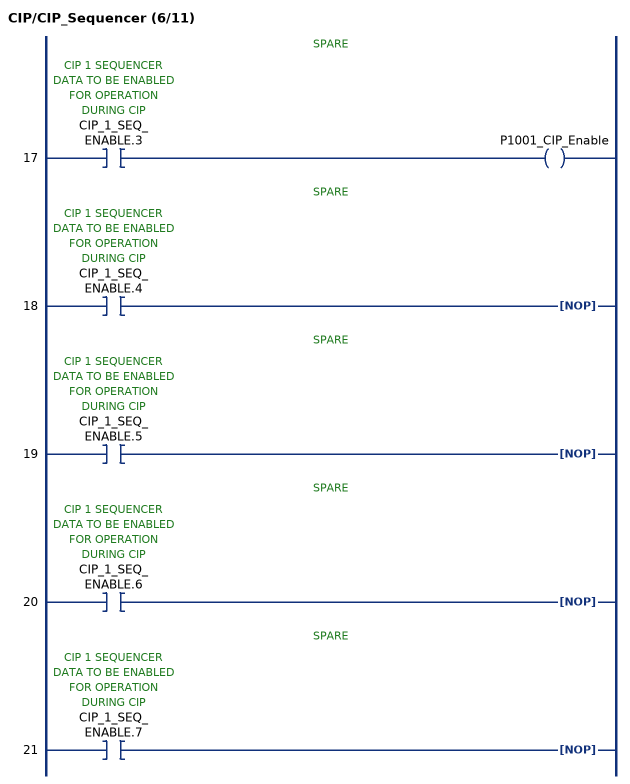
   // SPARE
   17: XIC(CIP_1_SEQ_ENABLE.3)OTE(P1001_CIP_Enable);
   // SPARE
   18: XIC(CIP_1_SEQ_ENABLE.4)NOP();
   // SPARE
   19: XIC(CIP_1_SEQ_ENABLE.5)NOP();
   // SPARE
   20: XIC(CIP_1_SEQ_ENABLE.6)NOP();
   // SPARE
   21: XIC(CIP_1_SEQ_ENABLE.7)NOP();
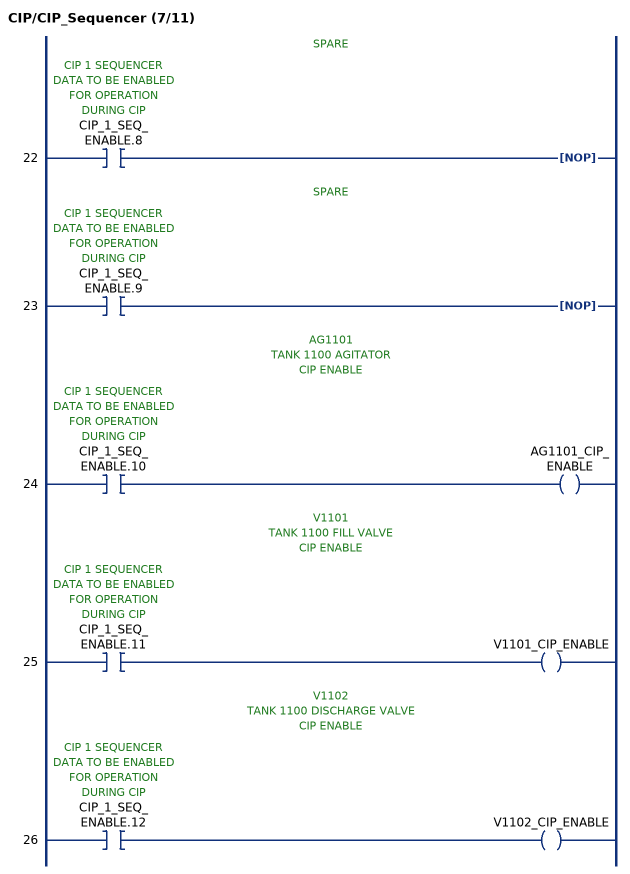
   // SPARE
   22: XIC(CIP_1_SEQ_ENABLE.8)NOP();
   // SPARE
   23: XIC(CIP_1_SEQ_ENABLE.9)NOP();
   // AG1101
   // TANK 1100 AGITATOR
   // CIP ENABLE
   24: XIC(CIP_1_SEQ_ENABLE.10)OTE(AG1101_CIP_ENABLE);
   // V1101
   // TANK 1100 FILL VALVE
   // CIP ENABLE
   25: XIC(CIP_1_SEQ_ENABLE.11)OTE(V1101_CIP_ENABLE);
   // V1102
   // TANK 1100 DISCHARGE VALVE
   // CIP ENABLE
   26: XIC(CIP_1_SEQ_ENABLE.12)OTE(V1102_CIP_ENABLE);
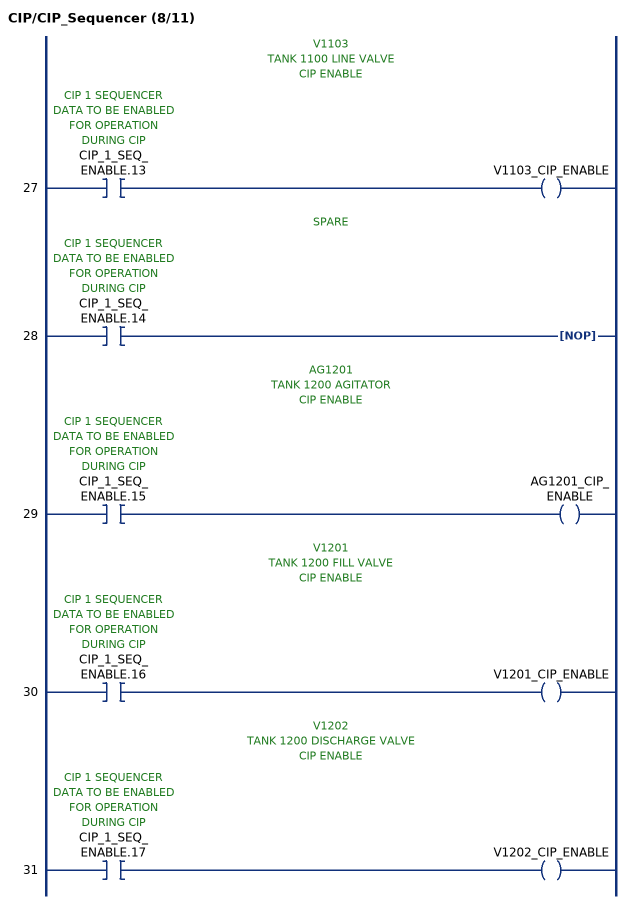
   // V1103
   // TANK 1100 LINE VALVE
   // CIP ENABLE
   27: XIC(CIP_1_SEQ_ENABLE.13)OTE(V1103_CIP_ENABLE);
   // SPARE
   28: XIC(CIP_1_SEQ_ENABLE.14)NOP();
   // AG1201
   // TANK 1200 AGITATOR
   // CIP ENABLE
   29: XIC(CIP_1_SEQ_ENABLE.15)OTE(AG1201_CIP_ENABLE);
   // V1201
   // TANK 1200 FILL VALVE
   // CIP ENABLE
   30: XIC(CIP_1_SEQ_ENABLE.16)OTE(V1201_CIP_ENABLE);
   // V1202
   // TANK 1200 DISCHARGE VALVE
   // CIP ENABLE
   31: XIC(CIP_1_SEQ_ENABLE.17)OTE(V1202_CIP_ENABLE);
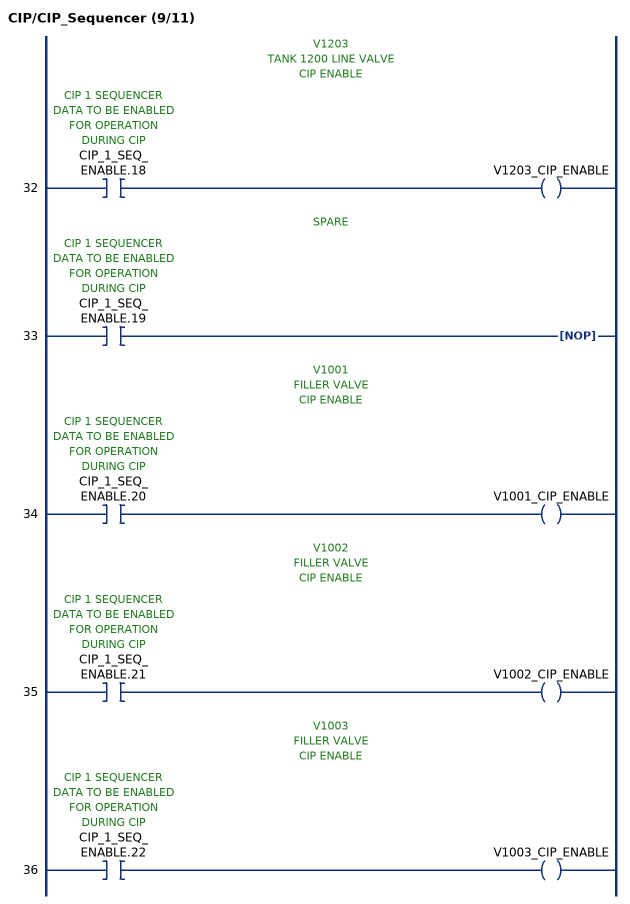
   // V1203
   // TANK 1200 LINE VALVE
   // CIP ENABLE
   32: XIC(CIP_1_SEQ_ENABLE.18)OTE(V1203_CIP_ENABLE);
   // SPARE
   33: XIC(CIP_1_SEQ_ENABLE.19)NOP();
   // V1001
   // FILLER VALVE
   // CIP ENABLE
   34: XIC(CIP_1_SEQ_ENABLE.20)OTE(V1001_CIP_ENABLE);
   // V1002
   // FILLER VALVE
   // CIP ENABLE
   35: XIC(CIP_1_SEQ_ENABLE.21)OTE(V1002_CIP_ENABLE);
   // V1003
   // FILLER VALVE
   // CIP ENABLE
   36: XIC(CIP_1_SEQ_ENABLE.22)OTE(V1003_CIP_ENABLE);
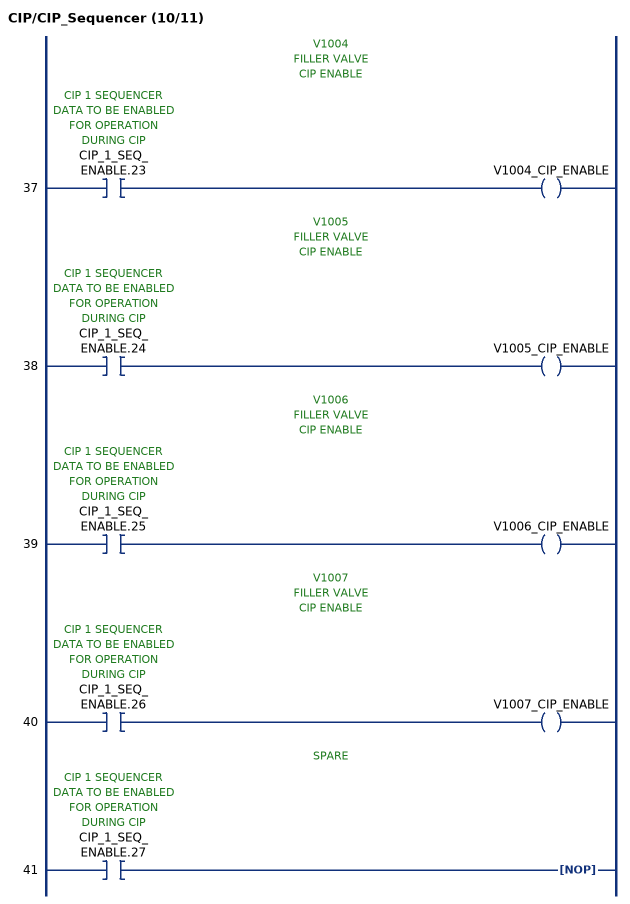
   // V1004
   // FILLER VALVE
   // CIP ENABLE
   37: XIC(CIP_1_SEQ_ENABLE.23)OTE(V1004_CIP_ENABLE);
   // V1005
   // FILLER VALVE
   // CIP ENABLE
   38: XIC(CIP_1_SEQ_ENABLE.24)OTE(V1005_CIP_ENABLE);
   // V1006
   // FILLER VALVE
   // CIP ENABLE
   39: XIC(CIP_1_SEQ_ENABLE.25)OTE(V1006_CIP_ENABLE);
   // V1007
   // FILLER VALVE
   // CIP ENABLE
   40: XIC(CIP_1_SEQ_ENABLE.26)OTE(V1007_CIP_ENABLE);
   // SPARE
   41: XIC(CIP_1_SEQ_ENABLE.27)NOP();
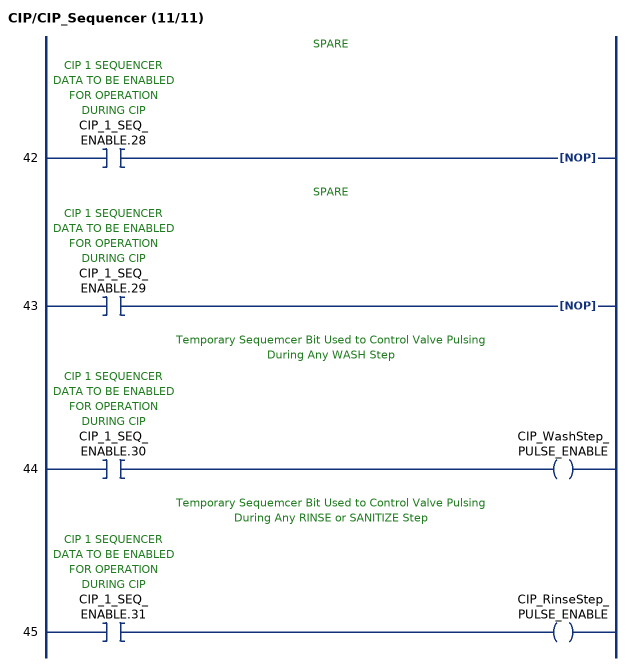
   // SPARE
   42: XIC(CIP_1_SEQ_ENABLE.28)NOP();
   // SPARE
   43: XIC(CIP_1_SEQ_ENABLE.29)NOP();
   // Temporary Sequemcer Bit Used to Control Valve Pulsing
   // During Any WASH Step
   44: XIC(CIP_1_SEQ_ENABLE.30)OTE(CIP_WashStep_PULSE_ENABLE);
   // Temporary Sequemcer Bit Used to Control Valve Pulsing
   // During Any RINSE or SANITIZE Step
   45: XIC(CIP_1_SEQ_ENABLE.31)OTE(CIP_RinseStep_PULSE_ENABLE);
END_ROUTINE
